FUNCTION_BLOCK TTestEventHandler_UsesEventArgs IMPLEMENTS ITestEventHandler_UsesEventArgs
VAR
    _EventWasRaised : BOOL;
    Arg1 : UDINT;
    Arg2 : LREAL;
    Arg3 : STRING;
    Arg4 : T_MAxString;
    Arg5 : BOOL;
END_VAR

PROPERTY EventWasRaised : BOOL
GET
EventWasRaised := _EventWasRaised;
END_GET
END_PROPERTY

METHOD OnThisEvent
VAR_INPUT
    EventArgs : IStreamReader;
END_VAR
Arg1 := EventArgs.Read_UDINT();
Arg2 := EventArgs.Read_LREAL();
Arg3 := EventArgs.Read_String();
Arg4 := EventArgs.Read_STRING();
Arg5 := EventArgs.Read_BOOL();

_EventWasRaised := TRUE;
END_METHOD

END_FUNCTION_BLOCK

(* stored: Version 1.1.0.1, ProductVersion 3.1.4024.4
   POU TTestEventHandler_UsesEventArgs: Id {87a28297-553f-4ed1-8c5d-366de471490c}, SpecialFunc None
   Property EventWasRaised: Id {aa467f9c-d09c-4800-a53a-09cdc5b8fd9d}
   Get Get: Id {8b7248f5-5871-424e-9c8a-ee967cc3826e}
   Method OnThisEvent: Id {7f79d98c-f159-43e7-b5ff-fd14bce07540} *)
